TYPE M2_location:
    (M2_A, M2_B);
END_TYPE

(* stored: ProductVersion 3.1.0.18, Version 1.1.0.1 *)
